PROGRAM main
VAR
	CAN_ERR : bool;
	K1_CAN_ON : bool;
	K2_CAN_ON : bool;
	K1_CAN_OFF : bool;
	K2_CAN_OFF : bool;
	BTN_ON_1 AT %IX0.3 : bool;
	BTN_ON_1_TMP : bool;
	BTN_ON_2 AT %IX0.5 : bool;
	BTN_ON_2_TMP : bool;
	K1 AT %QX0.0 : bool;
	K2 AT %QX0.1 : bool;
	BTN_OFF_1 AT %IX0.4 : bool;
	BTN_OFF_1_TMP : bool;
	BTN_OFF_2 AT %IX0.6 : bool;
	BTN_OFF_2_TMP : bool;
	CMD_WORD AT %MW0 : word;
	CYRCLE_STATE AT %MW1 : word := 0;
	TON0_TMP_ON : bool;
	TON1_TMP_ON : bool;
	TON2_TMP_ON : bool;
	TON3_TMP_ON : bool;
	CYCLE_RUN : bool;
	CYCLE_RUN_SET : bool;
	CMD_1 : bool;
	CMD_2 : bool;
	CMD_3 : bool;
	CMD_4 : bool;
	TON0 : TON;
	TON1 : TON;
	TON2 : TON;
	TON3 : TON;
	TON4 : TON;
	CAN_INTERFACE0 : CAN_INTERFACE;
	CAN_STATE AT %MW2 : word;
	BOOL_ON_WORD0 : BOOL_ON_WORD;
END_VAR
  VAR  (* added by the conversion: wires and edge detectors of the diagram *)
    _MOVE67_ENO : BOOL;
    _MOVE67_OUT : WORD;
    _MOVE77_ENO : BOOL;
    _MOVE77_OUT : WORD;
    _MOVE87_ENO : BOOL;
    _MOVE87_OUT : WORD;
    _MOVE97_ENO : BOOL;
    _MOVE97_OUT : WORD;
    _MOVE107_ENO : BOOL;
    _MOVE107_OUT : WORD;
    R_TRIG1 : R_TRIG;
    R_TRIG2 : R_TRIG;
    R_TRIG3 : R_TRIG;
    R_TRIG4 : R_TRIG;
    R_TRIG5 : R_TRIG;
    R_TRIG6 : R_TRIG;
  END_VAR

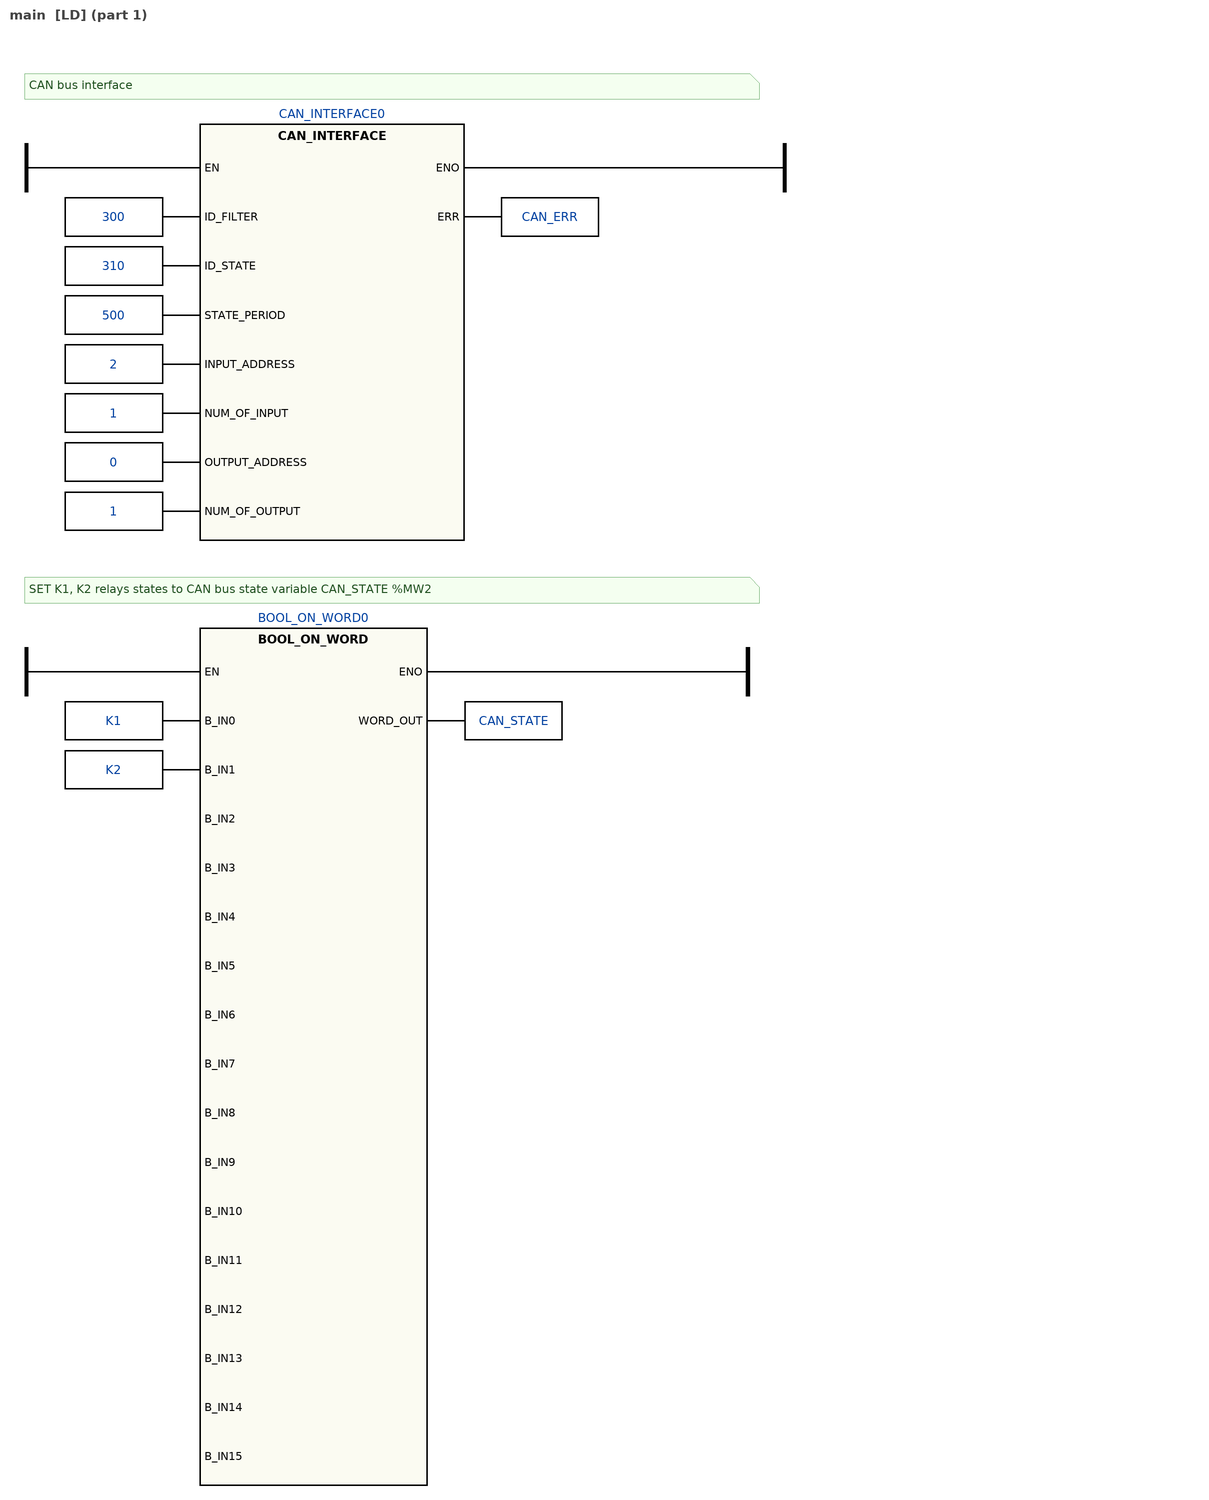
(* LD diagram, written out as Structured Text *)
(* CAN bus interface *)
CAN_INTERFACE0(ID_FILTER := 300, ID_STATE := 310, STATE_PERIOD := 500, INPUT_ADDRESS := 2, NUM_OF_INPUT := 1, OUTPUT_ADDRESS := 0, NUM_OF_OUTPUT := 1);
CAN_ERR := CAN_INTERFACE0.ERR;
(* SET K1, K2 relays states to CAN bus state variable CAN_STATE %MW2 *)
BOOL_ON_WORD0(B_IN0 := K1, B_IN1 := K2);
CAN_STATE := BOOL_ON_WORD0.WORD_OUT;
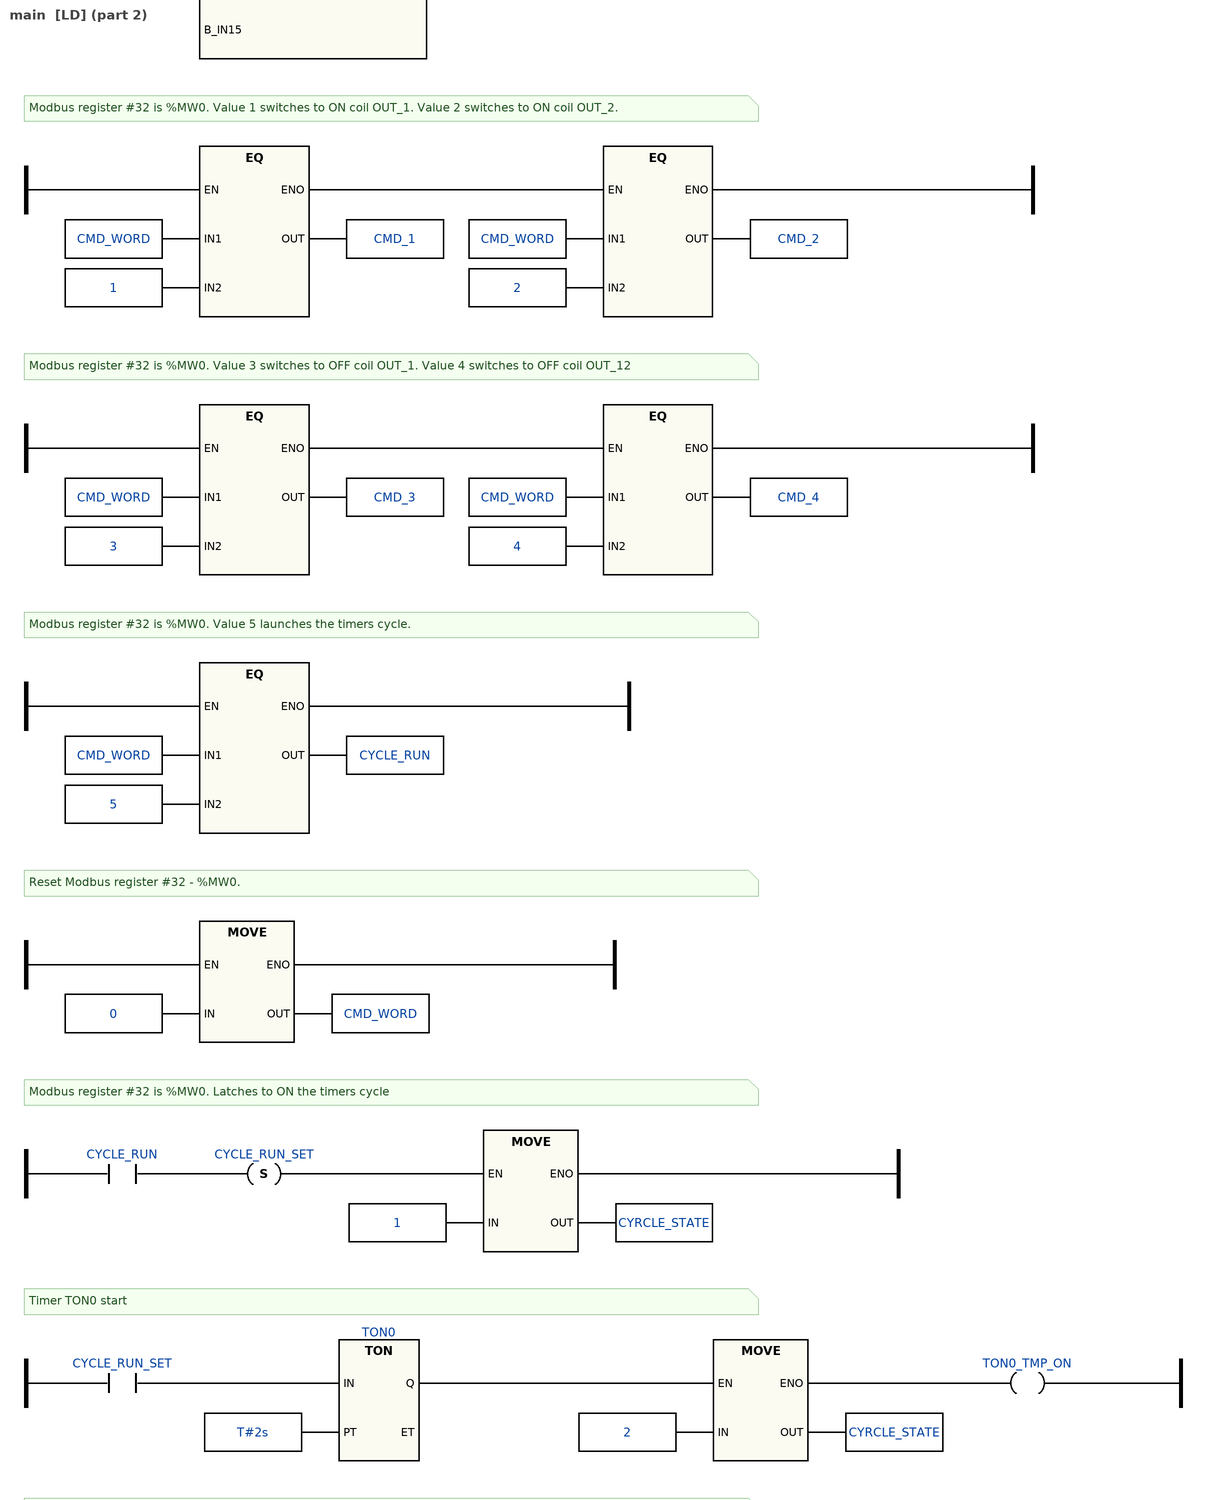
(* Modbus register #32 is %MW0. Value 1 switches to ON coil OUT_1. Value 2 switches to ON coil OUT_2. *)
CMD_1 := CMD_WORD = 1;
CMD_2 := CMD_WORD = 2;
(* Modbus register #32 is %MW0. Value 3 switches to OFF coil OUT_1. Value 4 switches to OFF coil OUT_12 *)
CMD_3 := CMD_WORD = 3;
CMD_4 := CMD_WORD = 4;
(* Modbus register #32 is %MW0. Value 5 launches the timers cycle. *)
CYCLE_RUN := CMD_WORD = 5;
(* Reset Modbus register #32 - %MW0. *)
CMD_WORD := 0;
(* Modbus register #32 is %MW0. Latches to ON the timers cycle *)
IF CYCLE_RUN THEN CYCLE_RUN_SET := TRUE; END_IF;
IF CYCLE_RUN THEN CYRCLE_STATE := 1; END_IF;
(* Timer TON0 start *)
TON0(IN := CYCLE_RUN_SET, PT := T#2s);
_MOVE67_OUT := MOVE(EN := TON0.Q, IN := 2, ENO => _MOVE67_ENO);
TON0_TMP_ON := _MOVE67_ENO;
IF _MOVE67_ENO THEN CYRCLE_STATE := _MOVE67_OUT; END_IF;
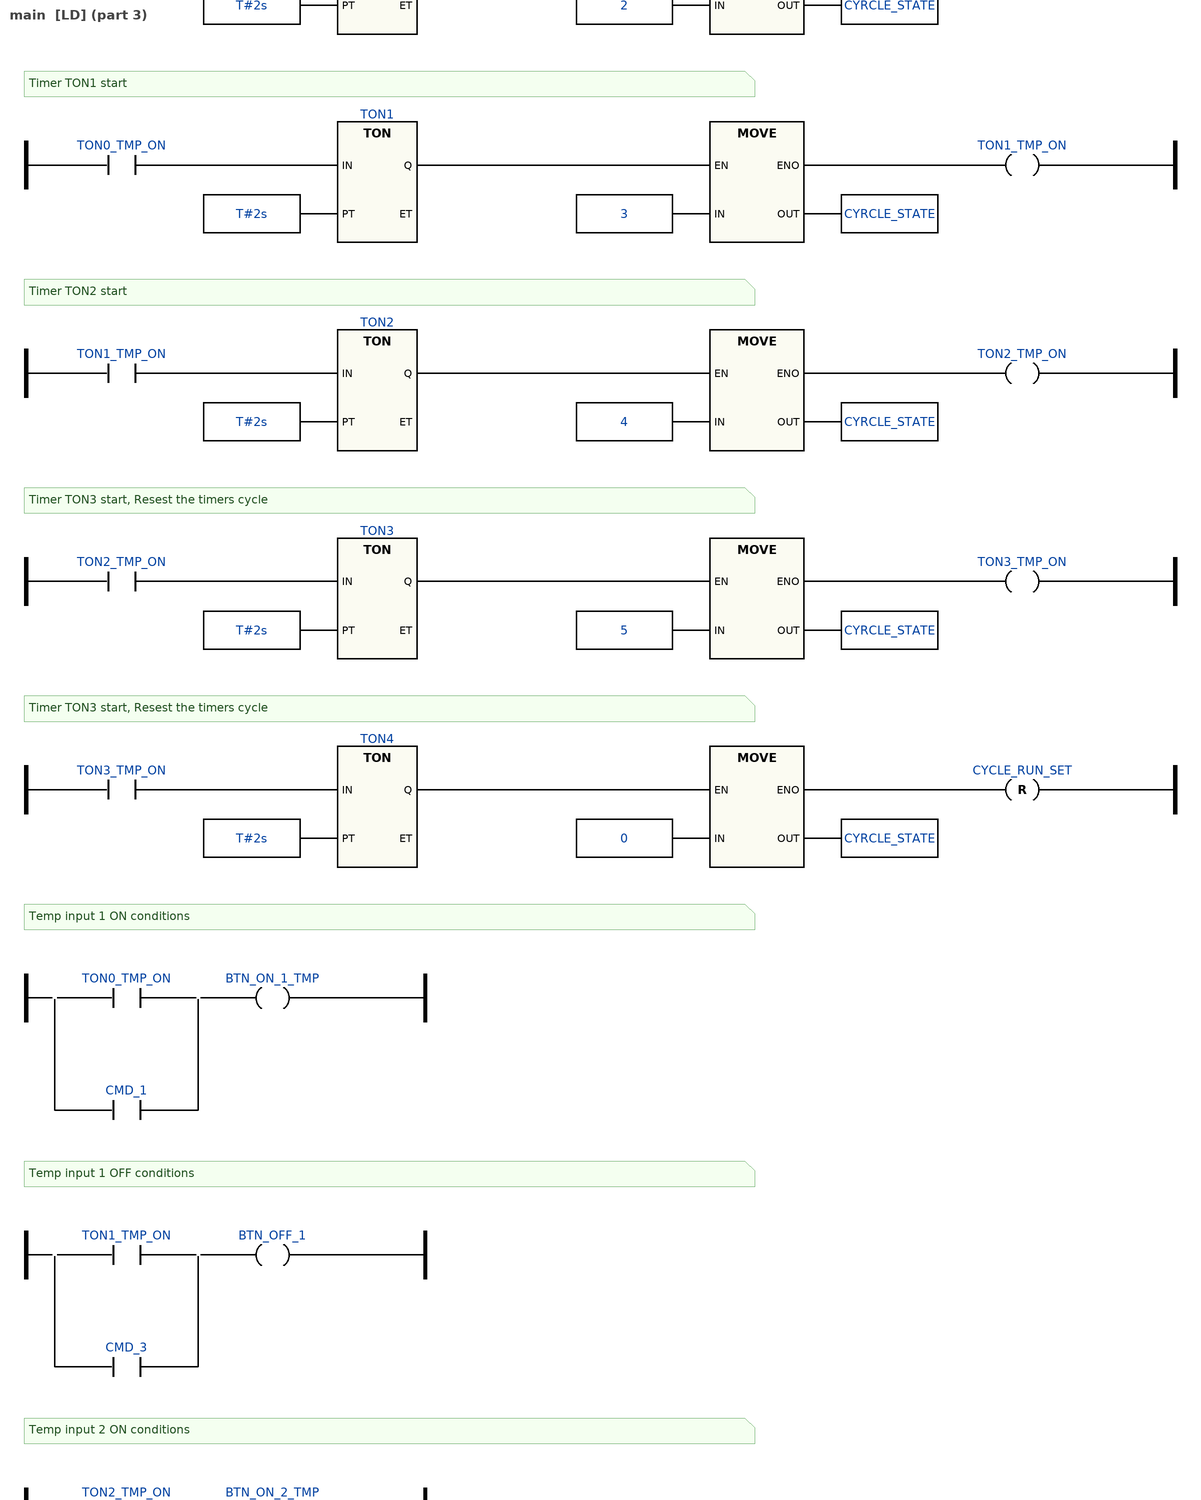
(* Timer TON1 start *)
TON1(IN := TON0_TMP_ON, PT := T#2s);
_MOVE77_OUT := MOVE(EN := TON1.Q, IN := 3, ENO => _MOVE77_ENO);
TON1_TMP_ON := _MOVE77_ENO;
IF _MOVE77_ENO THEN CYRCLE_STATE := _MOVE77_OUT; END_IF;
(* Timer TON2 start *)
TON2(IN := TON1_TMP_ON, PT := T#2s);
_MOVE87_OUT := MOVE(EN := TON2.Q, IN := 4, ENO => _MOVE87_ENO);
TON2_TMP_ON := _MOVE87_ENO;
IF _MOVE87_ENO THEN CYRCLE_STATE := _MOVE87_OUT; END_IF;
(* Timer TON3 start, Resest the timers cycle *)
TON3(IN := TON2_TMP_ON, PT := T#2s);
_MOVE97_OUT := MOVE(EN := TON3.Q, IN := 5, ENO => _MOVE97_ENO);
TON3_TMP_ON := _MOVE97_ENO;
IF _MOVE97_ENO THEN CYRCLE_STATE := _MOVE97_OUT; END_IF;
(* Timer TON3 start, Resest the timers cycle *)
TON4(IN := TON3_TMP_ON, PT := T#2s);
_MOVE107_OUT := MOVE(EN := TON4.Q, IN := 0, ENO => _MOVE107_ENO);
IF _MOVE107_ENO THEN CYCLE_RUN_SET := FALSE; END_IF;
IF _MOVE107_ENO THEN CYRCLE_STATE := _MOVE107_OUT; END_IF;
(* Temp input 1 ON conditions *)
BTN_ON_1_TMP := TON0_TMP_ON OR CMD_1;
(* Temp input 1 OFF conditions *)
BTN_OFF_1 := TON1_TMP_ON OR CMD_3;
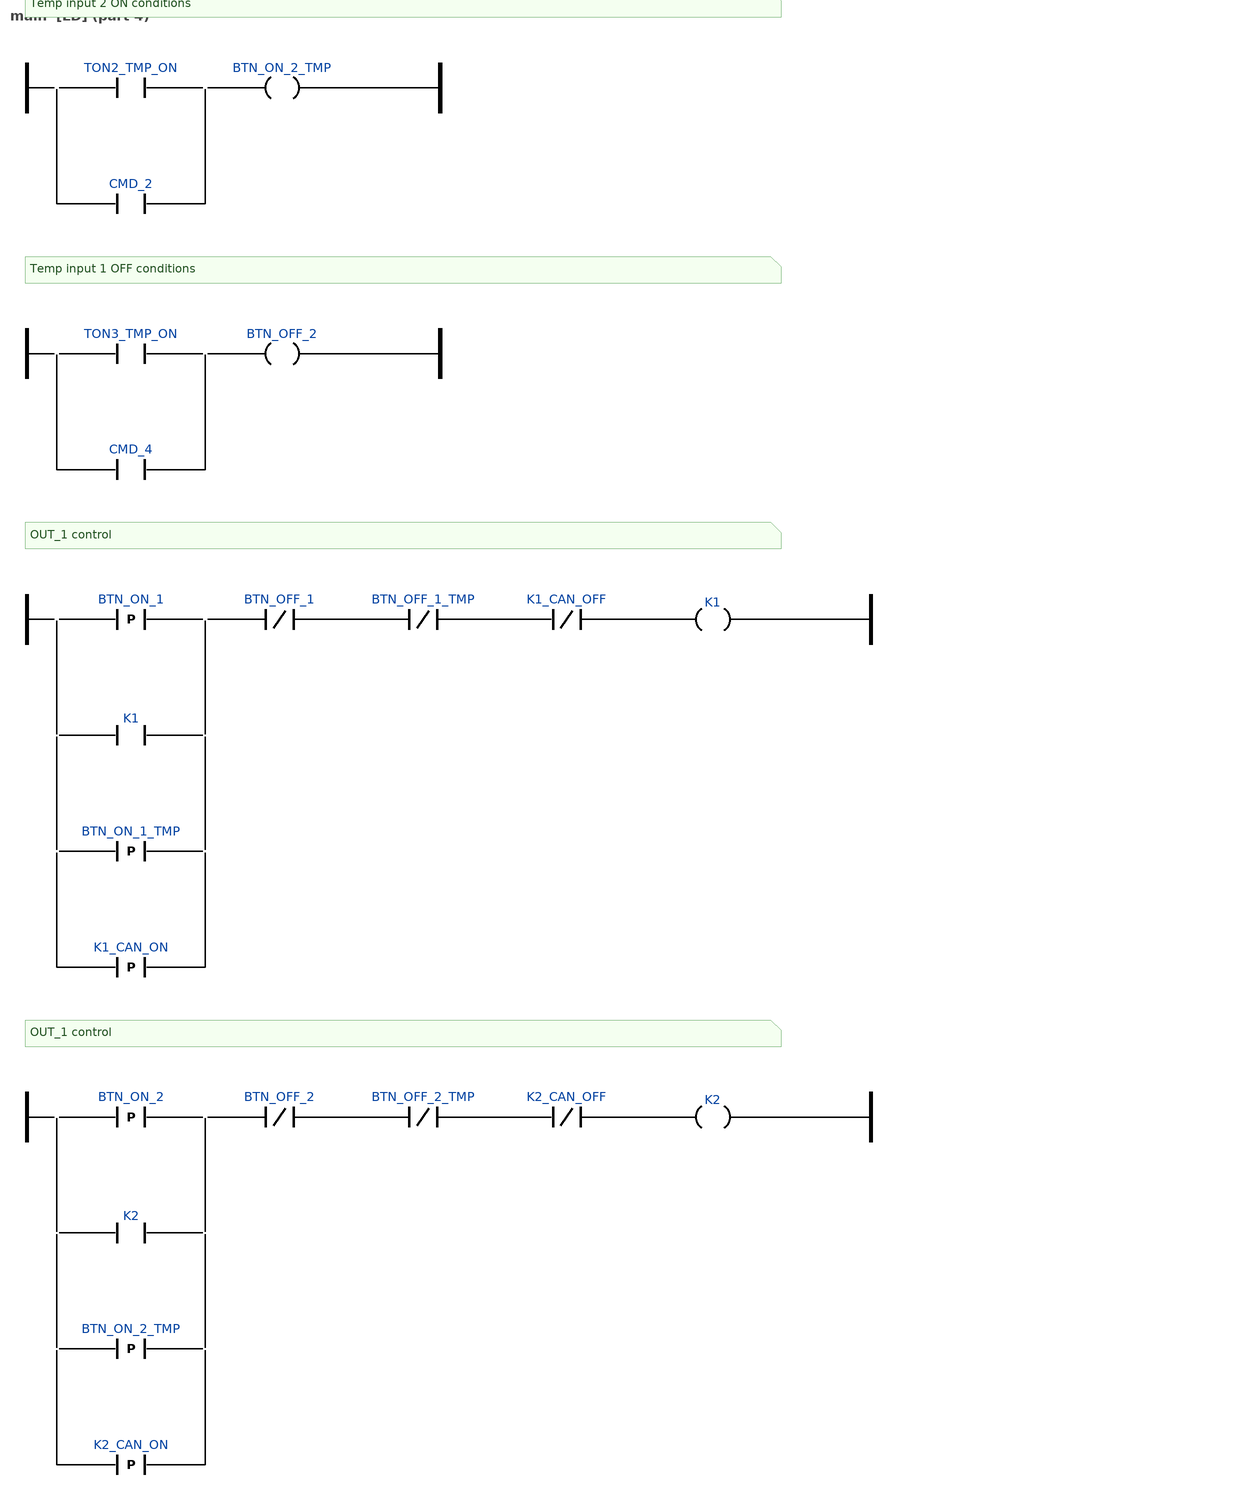
(* Temp input 2 ON conditions *)
BTN_ON_2_TMP := TON2_TMP_ON OR CMD_2;
(* Temp input 1 OFF conditions *)
BTN_OFF_2 := TON3_TMP_ON OR CMD_4;
(* OUT_1 control *)
R_TRIG1(CLK := BTN_ON_1);
R_TRIG2(CLK := BTN_ON_1_TMP);
R_TRIG3(CLK := K1_CAN_ON);
K1 := (R_TRIG1.Q OR K1 OR R_TRIG2.Q OR R_TRIG3.Q) AND NOT BTN_OFF_1 AND NOT BTN_OFF_1_TMP AND NOT K1_CAN_OFF;
(* OUT_1 control *)
R_TRIG4(CLK := BTN_ON_2);
R_TRIG5(CLK := BTN_ON_2_TMP);
R_TRIG6(CLK := K2_CAN_ON);
K2 := (R_TRIG4.Q OR K2 OR R_TRIG5.Q OR R_TRIG6.Q) AND NOT BTN_OFF_2 AND NOT BTN_OFF_2_TMP AND NOT K2_CAN_OFF;
END_PROGRAM
